PROGRAM prgComEffIO
VAR
	fbCom		: FB_MqttCommunicator_V2;
	
END_VAR


fbCom(
	bConnect:= TRUE, 
	strAuthKey:= 'EIO08031879806', 
	sUserName:= 'c0c17b06-0bdb-4698-a461-74f056a13e0b', 
	sUserPassword:= '80a8f7a1-49f9-455c-8c7e-584508cad010', 
	eSavePositionCertificate:= eSavePositionOnPLC.ePostionC,  
	time_HeartBeat_sec:= T#15S, 
	bConnected=> , 
	bError=> , 
	hrErrorCode=> , 
	eConnectionState=> , 
	eErrorMessage_Out=> );

END_PROGRAM

(* stored: Version 1.1.0.1, ProductVersion 3.1.4024.12
   POU prgComEffIO: Id {cbcd318b-bf51-484c-bcaa-d6efcdf43fe3}, SpecialFunc None *)
